SUBAPPLICATION Ventilsteuerung_Uebung_086 (* Beispiel für E_SWITCH *)
  (* Standard: 61499-2 *)
  (* Version 1.0, 2023-10-23, franz *)
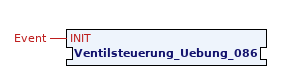
  EVENT_INPUT
    INIT;
  END_EVENT
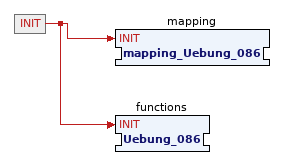
  SUBAPPS
    mapping : mapping_Uebung_086;
    functions : Uebung_086;
  END_SUBAPPS
  EVENT_CONNECTIONS
    INIT TO functions.INIT;
    INIT TO mapping.INIT;
  END_CONNECTIONS
END_SUBAPPLICATION
